(* CoDeSys 2.3.9.41 project: CTPowen150.pro *)
(* Libraries: STANDARD.LIB 4.10.05 11:14:46, IECSFC.LIB 13.4.06 15:51:28, SYSLIBTIME.LIB 20.2.06 13:31:16, SYSTASKINFO.LIB 20.2.06 13:31:38, ANALYZATION.LIB 5.10.99 09:05:06, SYSLIBCALLBACK.LIB 20.2.06 13:31:08 *)

(* PLC configuration (modules and I/O channels)
Discrete input 6 bit [ID100] node 0, in %IB0 out %QB0 {Filtrationtime = 10; Filtrationtime = 10; Filtrationtime = 10; Filtrationtime = 10; Filtrationtime = 10; Filtrationtime = 10; Visibility = No; PinCount = 6; WatchDogPeriod = 1000; PollPeriod = 1}
  AT %IX0.0 [BitInput]
  AT %IX0.1 [BitInput]
  AT %IX0.2 [BitInput]
  AT %IX0.3 [BitInput]
  AT %IX0.4 [BitInput]
  AT %IX0.5 [BitInput]
Discrete output 4 bit [ID101] node 1, in %IB1 out %QB1 {PinCount = 4; SafeValueBool = FALSE; SafeValueBool = FALSE; SafeValueBool = FALSE; SafeValueBool = FALSE; Visibility = No}
  AT %QX1.0 [BitOutput]
  AT %QX1.1 [BitOutput]
  AT %QX1.2 [BitOutput]
  AT %QX1.3 [BitOutput]
Special output [ID104] node 2, in %IB2 out %QB2 {Visibility = No; PinCount = 1}
  AT %QX2.0 [BitOutput] Special output
Unifed signal sensor [ID700] node 3, in %IB3 out %QB3 {Type_of_sensor700 = IT_0_20; measure_interval = 0.8; ainlow = 0; ainhigh = 20; first_cor_point = 0; first_delta = 0; second_cor_point = 0; second_delta = 0; third_cor_point = 0; third_delta = 0; Visibility = No}
  AT %ID3.0 [FloatInput] Value
  AT %IW3.1 [WordInput] Circular time
  Analog Input [ID107] node 0, in %IB3.0 out %QB3.0
Unifed signal sensor [ID700] node 4, in %IB4 out %QB4 {Type_of_sensor700 = IT_0_20; measure_interval = 0.8; ainlow = 0; ainhigh = 20; first_cor_point = 0; first_delta = 0; second_cor_point = 0; second_delta = 0; third_cor_point = 0; third_delta = 0; Visibility = No}
  AT %ID4.0 [FloatInput] Value
  AT %IW4.1 [WordInput] Circular time
  Analog Input [ID107] node 0, in %IB4.0 out %QB4.0
Unifed signal sensor [ID700] node 5, in %IB5 out %QB5 {Type_of_sensor700 = IT_0_20; measure_interval = 0.8; ainlow = 0; ainhigh = 20; first_cor_point = 0; first_delta = 0; second_cor_point = 0; second_delta = 0; third_cor_point = 0; third_delta = 0; Visibility = No}
  AT %ID5.0 [FloatInput] Value
  AT %IW5.1 [WordInput] Circular time
  Analog Input [ID107] node 0, in %IB5.0 out %QB5.0
Unifed signal sensor [ID700] node 6, in %IB6 out %QB6 {Type_of_sensor700 = IT_0_20; measure_interval = 0.8; ainlow = 0; ainhigh = 20; first_cor_point = 0; first_delta = 0; second_cor_point = 0; second_delta = 0; third_cor_point = 0; third_delta = 0; Visibility = No}
  AT %ID6.0 [FloatInput] Value
  AT %IW6.1 [WordInput] Circular time
  Analog Input [ID107] node 0, in %IB6.0 out %QB6.0
Analog output [ID106] node 7, in %IB7 out %QB7 {DAC_Type = Voltage 0-10 B; Analog_offset_correction = 0; Analog_full_range_correction = 0; SafeValueFloat = 0; Visibility = No}
  AT %QD7.0 [FloatOutput] Value
Analog output [ID106] node 8, in %IB8 out %QB8 {DAC_Type = Voltage 0-10 B; Analog_offset_correction = 0; Analog_full_range_correction = 0; SafeValueFloat = 0; Visibility = No}
  AT %QD8.0 [FloatOutput] Value
ModBus (Master) [MODBUS_MASTER_ID450] node 9, in %IB9 out %QB9 {Visibility = No}
  AT %QD9.0 [DWordOutput] Last address
  AT %QW9.1 [WordOutput] Last error
  RS-485-1 [COM1_USART] node 0, in %IB9.0 out %QB9.0 {CommunicationSpeed = 11520; Parity = NO PARITY CHECK; BitLength = 8 bits; StopLength = Two stop bits; InterfaceType = RS485; FrameOriented = RTU; Timeout = 0; Visibility = No}
AT %QB9.1.0 [ComChannel] Command (0xff - Start)
AT %IW9.1.0.0 [WordInput]
AT %IW9.1.1.0 [WordInput]
AT %QW9.1.2.0 [WordOutput]
AT %IW9.1.3.0 [WordInput]
Universal Modbus device [ID2000] node 2, in %IB9.2 out %QB9.2 {ModuleIP = 10:0:0:223; ServiceTimeout = 150; TCPport = 502; NetMode = Serial; ModuleSlaveAddress = 4; RequestType = By poll time; PeriodOfService = 3000; Visibility = No; RepeatCounter = 0; ByteSequence = Native}
  AT %QB9.2.0 [ComChannel] Command (0xff - Start)
AT %IW9.2.0.0 [WordInput]
AT %IW9.2.1.0 [WordInput]
AT %QW9.2.2.0 [WordOutput]
AT %IW9.2.3.0 [WordInput]
Universal Modbus device [ID2000] node 3, in %IB9.3 out %QB9.3 {ModuleIP = 10:0:0:223; ServiceTimeout = 150; TCPport = 502; NetMode = Serial; ModuleSlaveAddress = 5; RequestType = By poll time; PeriodOfService = 7000; Visibility = No; RepeatCounter = 0; ByteSequence = Trace_mode}
  AT %QB9.3.0 [ComChannel] Command (0xff - Start)
  32bit input module [ID2005] node 0, in %IB9.3.0 out %QB9.3.0 {ModbusAddress = 16009; Command_read_regs = Read holding Registers  (0x03); Visibility = No}
    AT %ID9.3.0.0 [DWordInput]
  32bit input module [ID2005] node 1, in %IB9.3.1 out %QB9.3.1 {ModbusAddress = 16099; Command_read_regs = Read holding Registers  (0x03); Visibility = No}
    AT %ID9.3.1.0 [DWordInput]
  Register input module [ID2003] node 2, in %IB9.3.2 out %QB9.3.2 {ModbusAddress = 16119; Command_read_regs = Read holding Registers  (0x03); Visibility = No}
    AT %IW9.3.2.0 [WordInput]
  Register input module [ID2003] node 3, in %IB9.3.3 out %QB9.3.3 {ModbusAddress = 16129; Command_read_regs = Read holding Registers  (0x03); Visibility = No}
    AT %IW9.3.3.0 [WordInput]
  32bit input module [ID2005] node 4, in %IB9.3.4 out %QB9.3.4 {ModbusAddress = 16139; Command_read_regs = Read holding Registers  (0x03); Visibility = No}
    AT %ID9.3.4.0 [DWordInput]
  32bit input module [ID2005] node 5, in %IB9.3.5 out %QB9.3.5 {ModbusAddress = 16519; Command_read_regs = Read holding Registers  (0x03); Visibility = No}
    AT %ID9.3.5.0 [DWordInput]
  32bit output module [ID2006] node 6, in %IB9.3.6 out %QB9.3.6 {ModbusAddress = 20209; Command_write_regs = Preset multiple Registers (0x10); Visibility = No}
    AT %QD9.3.6.0 [DWordOutput]
Debug RS-232 [DEBUG_USART] node 0, in %IB10.0.0 out %QB10.0.0 {CommunicationSpeed = 11520; Parity = EVEN; BitLength = 8 bits; StopLength = One stop bit; InterfaceType = RS232; FrameOriented = RTU; Timeout = 0; Visibility = No}
AT %QB10.1.0 [ByteOutput]
2 byte [Register] node 2, in %IB10.2 out %QB10.2
  AT %QW10.2.0 [WordOutput]
2 byte [Register] node 3, in %IB10.3 out %QB10.3
  AT %QW10.3.0 [WordOutput]
2 byte [Register] node 4, in %IB10.4 out %QB10.4
  AT %QW10.4.0 [WordOutput]
2 byte [Register] node 5, in %IB10.5 out %QB10.5
  AT %QW10.5.0 [WordOutput]
AT %QD10.6.0 [DWordOutput]
4 byte [FourBytes] node 7, in %IB10.7 out %QB10.7
  AT %QD10.7.0 [DWordOutput]
2 byte [Register] node 8, in %IB10.8 out %QB10.8
  AT %QW10.8.0 [WordOutput]
2 byte [Register] node 9, in %IB10.9 out %QB10.9
  AT %QW10.9.0 [WordOutput]
4 byte [FourBytes] node 10, in %IB10.10 out %QB10.10
  AT %QD10.10.0 [DWordOutput]
4 byte [FourBytes] node 11, in %IB10.11 out %QB10.11
  AT %QD10.11.0 [DWordOutput]
Archiver [ID650] node 11, in %IB11 out %QB11 {Archivation_mode = By timer; Archivation_type = ASCII only; Archivation_period = 360; Archive_name = CTP; Archive_version = trm1-trm2-fcP; Start_arch_time = Insert time in format HH:MM:SS; Stop_arch_time = Insert time in format HH:MM:SS; Arch_in_Sunday = Yes; Arch_in_Monday = Yes; Arch_in_Tuesday = Yes; Arch_in_Wednesday = Yes; Arch_in_Thursday = Yes; Arch_in_Friday = Yes; Arch_in_Saturday = Yes; Visibility = No}
  AT %QW11.0 [W32WordOutput] Status
  File output [FILE_Archivator] node 0, in %IB11.0 out %QB11.0 {Filename = CTP.log; FileWriteMode = Shift mode; FileType = Text; FileRecordsMaxCount = 4000; Visibility = No}
    AT %QW11.0.0 [WordOutput] File status
  16 bit [ID652] node 1, in %IB11.1 out %QB11.1 {Variable_name = GVS; Visibility = No}
    AT %QW11.1.0 [WordOutput]
  16 bit [ID652] node 2, in %IB11.2 out %QB11.2 {Variable_name = Insert variable name; Visibility = No}
    AT %QW11.2.0 [WordOutput]
  32 bit [ID653] node 3, in %IB11.3 out %QB11.3 {Variable_name = Insert variable name; Visibility = No}
    AT %QD11.3.0 [DWordOutput]
ModBus (slave) [MODBUS_ID400] node 12, in %IB12 out %QB12 {SlaveIdentificator = 1; Visibility = No}
  Modbus [MODBUS_ID302] node 0, in %IB12.0 out %QB12.0
    TCP [TCP_ID221] node 0, in %IB12.0.0 out %QB12.0.0 {RemotePort = 502; Visibility = No}
  2 byte [Register] node 1, in %IB12.1 out %QB12.1
    AT %QW12.1.0 [WordOutput]
  2 byte [Register] node 2, in %IB12.2 out %QB12.2
    AT %QW12.2.0 [WordOutput]
  2 byte [Register] node 3, in %IB12.3 out %QB12.3
    AT %QW12.3.0 [WordOutput]
  2 byte [Register] node 4, in %IB12.4 out %QB12.4
    AT %QW12.4.0 [WordOutput]
  2 byte [Register] node 5, in %IB12.5 out %QB12.5
    AT %QW12.5.0 [WordOutput]
  2 byte [Register] node 6, in %IB12.6 out %QB12.6
    AT %QW12.6.0 [WordOutput]
  2 byte [Register] node 7, in %IB12.7 out %QB12.7
    AT %QW12.7.0 [WordOutput]
  2 byte [Register] node 8, in %IB12.8 out %QB12.8
    AT %QW12.8.0 [WordOutput]
  4 byte [FourBytes] node 9, in %IB12.9 out %QB12.9
    AT %QD12.9.0 [DWordOutput]
  4 byte [FourBytes] node 10, in %IB12.10 out %QB12.10
    AT %QD12.10.0 [DWordOutput]
  4 byte [FourBytes] node 11, in %IB12.11 out %QB12.11
    AT %QD12.11.0 [DWordOutput]
  4 byte [FourBytes] node 12, in %IB12.12 out %QB12.12
    AT %QD12.12.0 [DWordOutput]
*)

(* Global variable list: Global_Variables *)
VAR_GLOBAL
(*ТРМ 1*)
	(*Состояние выхода*)
	Stat_Pan_1 AT %QX10.1.0.0 : BOOL;	(*передача на панель*)
	Stat_trm_1 AT %IW9.1.3.0 : WORD;	(*чтение с ТРМ'а*)

	(*температура и уставка*)
	T_panel1 AT %QW10.2.0 : WORD;
	T_trm1 AT %IW9.1.1.0 : WORD;
	Ts_panel1 AT %QW10.3.0 : WORD;
	Ts_trm1 AT %IW9.1.0.0 : WORD;

	(*задание уставки*)
	T_set1 AT %QW9.1.2.0 : WORD;

(*ТРМ 2*)
	(*Состояние выхода*)
	Stat_Pan_2 AT %QX10.1.0.1 : BOOL;	(*передача на панель*)
	Stat_trm_2 AT %IW9.2.3.0 : WORD;	(*чтение с ТРМ'а*)

	(*температура и уставка*)
	T_panel2 AT %QW10.4.0 : WORD;
	T_trm2 AT %IW9.2.1.0 : WORD;
	Ts_panel2 AT %QW10.5.0 : WORD;
	Ts_trm2 AT %IW9.2.0.0 : WORD;

	(*задание уставки*)
	T_set2 AT %QW9.2.2.0 : WORD;

(*задвижка*)
	Valve1 AT %QX10.1.0.2 : BOOL;
	Valve2 AT %QX10.1.0.3 : BOOL;

(*проверка связи*)
	Connection : INT;

(*пч*)
	(*для панели*)
	Ps_panel AT %QD10.6.0 : DWORD;
	Power_panel AT %QD10.7.0 : DWORD;
	Volt_panel AT %QW10.8.0 : WORD;
	Freq_panel AT %QW10.9.0 : WORD;
	Curr_panel AT %QD10.10.0 : DWORD;
	P_panel AT %QD10.11.0 : DWORD;

	(*с пч*)
	Ps_fc AT %ID9.3.0.0 : DWORD;
	Power_fc AT %ID9.3.1.0 : DWORD;
	Volt_fc AT %IW9.3.2.0 : WORD;
	Freq_fc AT %IW9.3.3.0 : WORD;
	Curr_fc AT %ID9.3.4.0 : DWORD;
	P_fc AT %ID9.3.5.0 : DWORD;

	(*на пч*)
	P_set AT %QD9.3.6.0 : DWORD;

(*архивы-архивчики*)
	T1_arch AT %QW11.1.0 : WORD;
	T2_arch AT %QW11.2.0 : WORD;
	P_arch AT %QD11.3.0 : DWORD;

(*delphi*)
	dT_trm1 AT %QW12.1.0 : WORD;
	dTs_trm1 AT %QW12.2.0 : WORD;
	dStat_trm_1 AT %QW12.3.0 : WORD;

	dT_trm2 AT %QW12.4.0 : WORD;
	dTs_trm2 AT %QW12.5.0 : WORD;
	dStat_trm_2 AT %QW12.6.0 : WORD;


	dVolt_fc AT %QW12.7.0 : WORD;
	dFreq_fc AT %QW12.8.0 : WORD;

	dPs_fc AT %QD12.9.0 : DWORD;
	dPower_fc AT %QD12.10.0 : DWORD;

	dCurr_fc AT %QD12.11.0 : DWORD;
	dP_fc AT %QD12.12.0 : DWORD;

END_VAR

(* POU PLC_PRG, ST *)
PROGRAM PLC_PRG
VAR
END_VAR
(*________ТРМ 1_________*)

(*передача ТРМ -> панель*)
T_panel1 := T_trm1;

(*изменение уставки*)
IF Ts_panel1 <> Ts_trm1
	THEN T_set1 := Ts_panel1;
END_IF;

(*состояние выхода*)
IF Stat_trm_1 = 1000
	THEN Stat_Pan_1 := 1;
		ELSE Stat_Pan_1 := 0;
END_IF;

(*_________ТРМ 2______*)

(*передача ТРМ -> панель*)
T_panel2 := T_trm2;

(*изменение уставки*)
IF Ts_panel2 <> Ts_trm2
	THEN T_set2 := Ts_panel2;
END_IF;

(*состояние выхода*)
IF Stat_trm_2 = 1000
	THEN Stat_Pan_2 := 1;
		ELSE Stat_Pan_2 := 0;
END_IF;

(*_______Задвижки______*)

IF Stat_Pan_1
	THEN Valve1 := 0;
		ELSE Valve1 := 1;
END_IF;

IF Stat_Pan_2
	THEN Valve2 := 0;
		ELSE Valve2 := 1;
END_IF;

(*_____Connection____*)
IF Connection=1
	THEN Connection := 2;
END_IF;

(*передача ПЧ -> панель*)
Power_panel := Power_fc;
Volt_panel := Volt_fc;
Freq_panel := Freq_fc;
Curr_panel := Curr_fc;
P_panel := P_fc;

(*задание уставки*)
IF Ps_panel <> Ps_fc
	THEN P_set := Ps_panel;
END_IF;


(*архивы-архивчики*)
T1_arch := T_trm1;
T2_arch := T_trm2;
P_arch :=	P_fc;


(*delphi*)
	dT_trm1 := T_trm1;
	dTs_trm1 := Ts_trm1;
	dStat_trm_1 := Stat_trm_1;

	dT_trm2 := T_trm2;
	dTs_trm2 := Ts_trm2;
	dStat_trm_2 := Stat_trm_2;


	dVolt_fc  := Volt_fc;
	dFreq_fc := Freq_fc;

	dPs_fc := Ps_fc;
	dPower_fc := Power_fc;

	dCurr_fc := Curr_fc;
	dP_fc := P_fc;
END_PROGRAM
